// TIA Portal V16 export
// export: Created 2022-11-01T21:54:09.7152714Z, ExportSetting WithDefaults, DisplayName Totally Integrated Automation Portal, DisplayVersion V16, DisplayName TIA Portal Version Control Interface, DisplayVersion V16, DisplayName TIA Portal Openness, DisplayVersion V16, DisplayName SINAMICS Startdrive Advanced, DisplayVersion V16, DisplayName SINAMICS Startdrive G130, G150, S120, S150, SINAMICS MV, S210, DisplayVersion V16, DisplayName SINAMICS Startdrive G110M, G120, G120C, G120D, G120P, DisplayVersion V16, DisplayName STEP 7 Professional, DisplayVersion V16, DisplayName STEP 7 Safety, DisplayVersion V16, DisplayName WinCC Professional, DisplayVersion V16
VAR_GLOBAL   // PLC tag table "AI C600-2"
   iTIR6101 AT %MW500 : Int;
   iTIR6102 AT %MW502 : Int;
   iTIR6103 AT %MW504 : Int;
   iTIR6104 AT %MW506 : Int;
   iTIR6105 AT %MW508 : Int;
   iTIR6106 AT %MW510 : Int;
   iTIR6107 AT %MW512 : Int;
   iTIR6108 AT %MW514 : Int;
   iTIR6109 AT %MW516 : Int;
   iTIR6110 AT %MW518 : Int;
   iTIR6111 AT %MW520 : Int;
   iTIR6112 AT %MW522 : Int;
   iTIR6113 AT %MW524 : Int;
   iTIR6114 AT %MW526 : Int;
   iTIR6115 AT %MW528 : Int;
   iTIR6116 AT %MW530 : Int;
   iTIR6117 AT %MW532 : Int;
   iTIR6118 AT %MW534 : Int;
   iTIR6120 AT %MW538 : Int;
   iTIR6121 AT %MW540 : Int;
   iTIR6123 AT %MW544 : Int;
   iTIR6124 AT %MW546 : Int;
   iTIR6125 AT %MW548 : Int;
   iTIR6126 AT %MW550 : Int;
   iTIR6127 AT %MW552 : Int;
   iTIR6128 AT %MW554 : Int;
   iTIR6129 AT %MW556 : Int;
   iTIR6130 AT %MW558 : Int;
   iTIR6133 AT %MW564 : Int;
   iTIR6134 AT %MW566 : Int;
   iTIR6135 AT %MW568 : Int;
   iTIR6137 AT %MW572 : Int;
   iTIR6138 AT %MW574 : Int;
   iTIR6139 AT %MW576 : Int;
   iTIR6141 AT %MW580 : Int;
   iTIR6142 AT %MW582 : Int;
   iTIR6143 AT %MW584 : Int;
   iTIR6144 AT %MW586 : Int;
   iTIR6145 AT %MW588 : Int;
   iTIR6146 AT %MW590 : Int;
   iTIR6147 AT %MW592 : Int;
   iTIR6149 AT %MW596 : Int;
   iTIR6150 AT %MW598 : Int;
   iTIR6151 AT %MW600 : Int;
   iTIR6152 AT %MW602 : Int;
   iTIR6153 AT %MW604 : Int;
   iTIR6154 AT %MW606 : Int;
   iTIR6155 AT %MW608 : Int;
   iTIR6156 AT %MW610 : Int;
   iTIR6157 AT %MW612 : Int;
   iTIR6158 AT %MW614 : Int;
   iTIR6159 AT %MW616 : Int;
   iTIR6160 AT %MW618 : Int;
   iTIR6161 AT %MW620 : Int;
   iTIR6162 AT %MW622 : Int;
   iTIR6163 AT %MW624 : Int;
   iTIR6164 AT %MW626 : Int;
   iTIR6165 AT %MW628 : Int;
   iTIR6166 AT %MW630 : Int;
   iTIR6167 AT %MW632 : Int;
   iTIR6168 AT %MW634 : Int;
   iTIR6169 AT %MW636 : Int;
   iTIR6170 AT %MW638 : Int;
   iTIR6171 AT %MW640 : Int;
   iTIR6172 AT %MW642 : Int;
   iTIR6173 AT %MW644 : Int;
   iTIR6174 AT %MW646 : Int;
   iTIR6175 AT %MW648 : Int;
   iTIR6176 AT %MW650 : Int;
   iTIR6177 AT %MW652 : Int;
   iTIR6178 AT %MW654 : Int;
   iTIR6179 AT %MW656 : Int;
   iTIR6180 AT %MW658 : Int;
   iTIR6181 AT %MW660 : Int;
   iTIR6182 AT %MW662 : Int;
   iQIR6101 AT %MW664 : Int;
   iQIR6102 AT %MW666 : Int;
   iQIR6103 AT %MW668 : Int;
   iQIR6104 AT %MW670 : Int;
   iTIR6119 AT %MW536 : Int;
   iTIR6122 AT %MW542 : Int;
   iTIR6131 AT %MW560 : Int;
   iTIR6132 AT %MW562 : Int;
   iTIR6136 AT %MW570 : Int;
   iTIR6140 AT %MW578 : Int;
   iTIR6148 AT %MW594 : Int;
   iPIR6101 AT %MW672 : Int;
   iPIR6102 AT %MW674 : Int;
   iPIR6103 AT %MW676 : Int;
   iPIR6104 AT %MW678 : Int;
   iPIR6105 AT %MW680 : Int;
   iPIR6106 AT %MW682 : Int;
   iPIR6107 AT %MW684 : Int;
   iPIR6108 AT %MW686 : Int;
   iPIR6109 AT %MW688 : Int;
   iPIR6110_virtual AT %MW690 : Int;
   iPIR6111 AT %MW692 : Int;
   iPIR6112 AT %MW694 : Int;
   iPIR6113_virtual AT %MW696 : Int;
   iPIR6114 AT %MW698 : Int;
   iPIR6115 AT %MW700 : Int;
   iPIR6116_virtual AT %MW702 : Int;
   iPIR6117 AT %MW704 : Int;
   iPIR6118 AT %MW706 : Int;
   iPIR6119 AT %MW708 : Int;
   iPIR6120 AT %MW710 : Int;
   iPIR6121 AT %MW712 : Int;
   iPIR6122 AT %MW714 : Int;
   iPIR6123 AT %MW716 : Int;
   iPIR6124 AT %MW718 : Int;
   iPIR6125 AT %MW720 : Int;
   iPIR6126 AT %MW722 : Int;
   iPIR6127 AT %MW724 : Int;
   iPIR6128 AT %MW726 : Int;
   iPIR6129 AT %MW728 : Int;
   iPIR6130 AT %MW730 : Int;
   iPIR6131 AT %MW732 : Int;
   iPIR6132 AT %MW734 : Int;
   iPIR6133 AT %MW736 : Int;
   iPIR6134 AT %MW738 : Int;
   iPIR6135 AT %MW740 : Int;
   iPIR6136 AT %MW742 : Int;
   iPIR6137 AT %MW744 : Int;
   iPIR6138 AT %MW746 : Int;
   iPIR6139 AT %MW748 : Int;
   iPIR6140 AT %MW750 : Int;
   iPIR6141 AT %MW752 : Int;
   iPIR6142 AT %MW754 : Int;
   iPIR6143 AT %MW756 : Int;
   iPIR6144 AT %MW758 : Int;
   iPIR6145 AT %MW760 : Int;
   iPIR6146 AT %MW762 : Int;
   iPIR6147 AT %MW764 : Int;
   iPIR6148 AT %MW766 : Int;
   iPIR6149 AT %MW768 : Int;
   iPIR6150 AT %MW770 : Int;
   iPIR6151 AT %MW772 : Int;
   iLIR6101 AT %MW774 : Int;
   iLIR6102 AT %MW776 : Int;
   iLIR6103 AT %MW778 : Int;
   iLIR6104 AT %MW780 : Int;
   iLIR6105 AT %MW782 : Int;
   iLIR6106 AT %MW784 : Int;
   iLIR6107 AT %MW786 : Int;
   iLIR6108 AT %MW788 : Int;
   iLIR6109 AT %MW790 : Int;
   iLIR6110 AT %MW792 : Int;
   iLIR6111 AT %MW794 : Int;
   iLIR6112 AT %MW796 : Int;
   iLIR6113 AT %MW798 : Int;
   iLIR6114 AT %MW800 : Int;
   iLIR6115 AT %MW802 : Int;
   iLIR6116 AT %MW804 : Int;
   iLIR6117 AT %MW806 : Int;
   iLIR6118 AT %MW808 : Int;
   iLIR6119 AT %MW810 : Int;
   iLIR6120 AT %MW812 : Int;
   iLIR6121 AT %MW814 : Int;
   iLIR6122 AT %MW816 : Int;
   iLIR6123 AT %MW818 : Int;
   iFIR6101 AT %MW820 : Int;
   iFIR6102 AT %MW822 : Int;
   iFIR6103 AT %MW824 : Int;
   iFIR6104 AT %MW826 : Int;
   iFIR6105 AT %MW828 : Int;
   iFIR6106 AT %MW830 : Int;
   iFIR6107 AT %MW832 : Int;
   iFIR6108 AT %MW834 : Int;
   iFIR6109 AT %MW836 : Int;
   iFIR6110 AT %MW838 : Int;
   iFIR6111 AT %MW840 : Int;
   iFIR6112 AT %MW842 : Int;
   iFIR6113 AT %MW844 : Int;
   iFIR6114 AT %MW846 : Int;
   iFIR6115 AT %MW848 : Int;
   iFIR6116 AT %MW850 : Int;
   iFIR6117 AT %MW852 : Int;
   iFIR6118 AT %MW854 : Int;
   iFIR6119 AT %MW856 : Int;
   iFIR6120 AT %MW858 : Int;
   iFIR6121 AT %MW860 : Int;
   iFIR6122 AT %MW862 : Int;
   iFIR6123 AT %MW864 : Int;
   "iFIR6115-1" AT %MW866 : Int;
END_VAR
